{attribute 'qualified_only'}
VAR_GLOBAL
END_VAR

(* stored: Version 1.1.0.1, ProductVersion 3.1.4024.12
   GVL G_Output: Id {31e18101-edb6-4be0-8891-f5a4461ec477} *)
